// TIA Portal project "G INVERSION DE GIRO" (V11)

(* hardware
DEVICE "S7300/ET200 station_1"  SIMATIC 300-Station
   slot 0: "Perfil soporte_0"  Rail  6ES7 390-1***0-0AA0
   slot 2: "PLC_1"  CPU 313C-2 DP  6ES7 313-6CF03-0AB0  V2.6
      slot 0: "Interfaz MPI_1"  MPI
      slot 1: "Interfaz DP_1"  DP
      slot 2: "DI16/DO16_1"  DI16/DO16
      slot 4: "Contaje_1"  Counter
*)

// ===== PLC "PLC_1"  CPU 313C-2 DP =====

VAR_GLOBAL   // PLC tag table "Tabla de variables estándar"
   "Tag_1" AT %A0.0 : Bool;
   "Tag_2" AT %A0.1 : Bool;
   "Tag_3" AT %A0.2 : Bool;
   "Tag_4" AT %E0.0 : Bool;
   "Tag_5" AT %E0.1 : Bool;
   "Tag_6" AT %E0.2 : Bool;
   "Tag_7" AT %T0 : Timer;
   "Tag_8" AT %M0.0 : Bool;
END_VAR

DATA_BLOCK "INVERSION DE GIRO_DB"   // DB1
{ S7_Optimized_Access := 'FALSE' }
VERSION : 0.1
// stored: InstanceOfName INVERSION DE GIRO
"INVERSION DE GIRO"
BEGIN
   SWITCH[0] := 16#0;
   SW_SQTS[0] := 16#3;
   SW_SQTS[1] := 16#0;
   SW_SQTS[2] := 16#1;
   SW_SQTS[3] := 16#2;
   TVX[0] := 16#1;
   TTX[0] := 16#1;
   TSX[0] := 16#1;
   S00X[0] := 16#1;
   SOFFX[0] := 16#1;
   SONX[0] := 16#1;
   SAX[0] := 16#1;
   SERRX[0] := 16#1;
   SMX[0] := 16#1;
   S0X[0] := 16#1;
   S1X[0] := 16#1;
   SINI[0] := 16#2;
   SINI[1] := 16#1;
   LSTT[3] := 16#1;
   LSTT[4] := 16#1;
   ATAJ[1] := 16#1;
   ATAJ[2] := 16#2;
   ATAJ[3] := 16#3;
   ATAJ[4] := 16#4;
   ATAB[1] := 16#2;
   ATAB[2] := 16#1;
   ATAB[3] := 16#3;
   ATAB[4] := 16#4;
   PSTT[1] := 16#1;
   PSTT[2] := 16#1;
   PSTT[3] := 16#2;
   PSTT[4] := 16#3;
   NSTT[0] := 16#1;
   NSTT[1] := 16#2;
   NSTT[2] := 16#3;
   NSTT[3] := 16#1;
   NSTT[4] := 16#1;
   ASSJ[1] := 16#1;
   ASSJ[2] := 16#2;
   ASSJ[3] := 16#3;
   ASSB[1] := 16#1;
   ASSB[2] := 16#2;
   ASSB[3] := 16#3;
   PTTS[1] := 16#0;
   PTTS[2] := 16#1;
   PTTS[3] := 16#2;
   NTTS[1] := 16#1;
   NTTS[2] := 16#3;
   NTTS[3] := 16#4;
END_DATA_BLOCK

FUNCTION_BLOCK "INVERSION DE GIRO"   // FB1, GRAPH
{ S7_Optimized_Access := 'FALSE' }
VERSION : 0.1
   VAR_INPUT
      OFF_SQ : Bool := false;   // Desconectar cadena
      INIT_SQ : Bool := false;   // Poner cadena en estado inicial
      ACK_EF : Bool := false;   // Acusar todos los errores y fallos
      S_PREV : Bool := false;   // Mostrar la etapa anterior en el parámetro S_NO
      S_NEXT : Bool := false;   // Mostrar la etapa siguiente en el parámetro S_NO
      SW_AUTO : Bool := false;   // Modo automático
      SW_TAP : Bool := false;   // Semiautomático/continuar con transición
      SW_TOP : Bool := false;   // Semiautomático/transición ignorada
      SW_MAN : Bool := false;   // Modo manual
      S_SEL : Int := 0;   // Seleccionar la etapa que debe mostrarse en S_NO
      S_ON : Bool := false;   // Activar la etapa del parámetro S_NO
      S_OFF : Bool := false;   // Desactivar el incremento presente en el parámetro S_NO
      T_PUSH : Bool := false;   // Habilitar transición en modo semiautomático
      "MARCHA DERECHA" : Bool;
      "MARCHA IZQUIERDA" : Bool;
      PARO : Bool;
   END_VAR
   VAR_OUTPUT
      S_NO : Int := 0;   // Número de etapa
      S_MORE : Bool := false;   // Existen más etapas que pueden mostrarse en S_NO.
      S_ACTIVE : Bool := false;   // El incremento presente en el parámetro S_NO está activo
      ERR_FLT : Bool := false;   // Error de grupo interlock o supervisión
      AUTO_ON : Bool := false;   // Modo automático activado
      TAP_ON : Bool := false;   // Modo semiautomático/etapa con transición activada
      TOP_ON : Bool := false;   // Modo semiautomático/Ignorar transición activado
      MAN_ON : Bool := false;   // Modo manual activado
      "GIRO DERECHA" : Bool;
      "GIRO IZQUIERDA" : Bool;
   END_VAR
   VAR
      SWITCH : Array [0..0]of DWord;
      SW_SQTS : Array [0..3]of Byte;
      SW_ADDR : Word := 16#A;
      G7T_0 : GraphTransition;
      DERECHA : GraphTransition;
      IZQUIERDA : GraphTransition;
      "PARO D" : GraphTransition;
      "PARO I" : GraphTransition;
      G7S_0 : GraphStep;
      REPOSO : GraphStep;
      "M.D." : GraphStep;
      "M.I." : GraphStep;
      PRE_CRIT : Array [0..0]of DWord;
      POST_CRIT : Array [0..0]of DWord;
      TVX : Array [0..4]of Byte;
      TTX : Array [0..4]of Byte;
      TSX : Array [0..2]of Byte;
      S00X : Array [0..2]of Byte;
      SOFFX : Array [0..2]of Byte;
      SONX : Array [0..2]of Byte;
      SAX : Array [0..2]of Byte;
      SERRX : Array [0..4]of Byte;
      SMX : Array [0..4]of Byte;
      S0X : Array [0..4]of Byte;
      S1X : Array [0..4]of Byte;
      S_DISPLAY : Int;   // Indicación interna del parámetro de salida S_NO
      S_SEL_OLD : Int;   // Valor anterior en S_SEL
      S_DISPIDX : Byte;   // Índice de la etapa presente en S_NO
      T_DISPIDX : Byte;   // Índice de la transición presente en T_NO
      MOPEDGE : Struct
         AUTO : Bool := false;
         MAN : Bool := false;
         TAP : Bool := false;
         TOP : Bool := false;
         ACK_S : Bool := false;
         REG_S : Bool := false;
         T_PREV : Bool := false;
         T_NEXT : Bool := false;
         LOCK : Bool := false;
         SUP : Bool := false;
         ACKREQ : Bool := false;
         SSKIP : Bool := false;
         OFF : Bool := false;
         INIT : Bool := false;
         HALT : Bool := false;
         TMS_HALT : Bool := false;
         OPS_ZERO : Bool := false;
         SACT_DISP : Bool := false;
         SEF_DISP : Bool := false;
         SALL_DISP : Bool := false;
         S_PREV : Bool := false;
         S_NEXT : Bool := false;
         S_SELOK : Bool := false;
         S_ON : Bool := false;
         S_OFF : Bool := false;
         T_PUSH : Bool := false;
         REG : Bool := false;
         ACK : Bool := false;
         IL_PERM : Bool := false;
         T_PERM : Bool := false;
         ILP_MAN : Bool := false;
      END_STRUCT;
      MOP : Struct   // Modo de operación
         AUTO : Bool := true;   // Estado: modo automático
         MAN : Bool := false;   // Estado: modo manual
         TAP : Bool := false;   // Estado: semiautomático/continuar con transición
         TOP : Bool := false;   // Estado: semiautomático/transición ignorada
         ACK_S : Bool := false;   // Solicitud: acusar la etapa presente en el parámetro S_NO
         REG_S : Bool := false;   // Solicitud: registrar la etapa presente en el parámetro S_NO
         T_PREV : Bool := false;   // Solicitud: mostrar la transición anterior válida en el parámetro T_NO
         T_NEXT : Bool := false;   // Solicitud: mostrar la siguiente transición válida en el parámetro T_NO
         LOCK : Bool := true;   // Estado: ejecución de interlock activada
         SUP : Bool := true;   // Estado: ejecución de supervisión activada
         ACKREQ : Bool := true;   // Estado: acuse requerido
         SSKIP : Bool := false;   // Estado: "Saltar etapas" activado
         OFF : Bool := false;   // Solicitud: desactivar todas las etapas
         INIT : Bool := true;   // Solicitud: poner cadena en estado inicial
         HALT : Bool := false;   // Estado: la cadena no continúa
         TMS_HALT : Bool := false;   // Estado: todos los temporizadores internos detenidos
         OPS_ZERO : Bool := false;   // Estado: todos los operandos ejecutados con N, L, D puestos a 0
         SACT_DISP : Bool := true;   // Estado: mostrar sólo etapas activas
         SEF_DISP : Bool := false;   // Estado: mostrar sólo etapas erróneas y defectuosas
         SALL_DISP : Bool := false;   // Estado: mostrar todas las etapas
         S_PREV : Bool := false;   // Solicitud: mostrar la etapa anterior en el parámetro S_NO
         S_NEXT : Bool := false;   // Solicitud: Indicar etapa siguiente en el parámetro S_NO
         S_SELOK : Bool := false;   // Solicitud: mostrar en el parámetro S_NO el número de la etapa presente en el parámetro S_SEL
         S_ON : Bool := false;   // Solicitud: activar la etapa presente en el parámetro S_NO
         S_OFF : Bool := false;   // Solicitud: desactivar la etapa presente en el parámetro S_NO
         T_PUSH : Bool := false;   // Solicitud: habilitar transición
         REG : Bool := false;   // Solicitud: registrar todos los errores de interlock y supervisión
         ACK : Bool := false;   // Solicitud: acusar todos los errores de interlock y supervisión
         IL_PERM : Bool := false;   // Estado: ejecución permanente de todos los interlocks
         T_PERM : Bool := false;   // Estado: ejecución permanente de todas las transiciones
         ILP_MAN : Bool := false;   // Estado: ejecución permanente de todos los interlocks en modo manual
      END_STRUCT;
      TICKS : Struct   // Ciclos de tiempo
         DELTA : Time := T#0ms;   // Diferencia de tiempo entre dos ciclos
         OLD : Time := T#0ms;   // Estado de contador cíclico 10 ms en el último ciclo
         NEW : Time := T#0ms;   // Estado de contador cíclico 10 ms en este ciclo
      END_STRUCT;
      SQ_FLAGS : Struct   // Marcas de cadena
         ERR_FLT : Bool := false;   // Error de grupo interlock y supervisión
         ERROR : Bool := false;   // Error de grupo Interlock
         FAULT : Bool := false;   // Error de grupo Supervisión
         RT_FAIL : Bool := false;   // Error en tiempo de ejecución
         NO_SNO : Bool := false;   // No se ha encontrado el número de etapa solicitado
         NF_OFL : Bool := false;   // Desbordamiento: demasiadas solicitudes ON u OFF
         SA_OFL : Bool := false;   // Desbordamiento: demasiadas etapas activas
         TV_OFL : Bool := false;   // Desbordamiento: demasiadas transiciones válidas
         MSG_OFL : Bool := false;   // Desbordamiento: los recursos del sistema no son suficientes para ALARM_S
         NO_SWI : Bool := false;   // No conmutar en este ciclo
         CYC_OP : Bool := false;   // Ejecución cíclica de la cadena tras la inicialización
         AS_MSG : Bool := true;   // Avisos en tiempo de ejecución activados o desactivados por instrucción
         AS_SEND : Bool := false;   // Enviar avisos de WR_USMSG o sólo registrarlos en el búfer de diagnóstico
         SQ_BUSY : Bool := false;   // Marca de flanco interna para ejecución de proceso
         SA_BUSY : Bool := false;   // Marca de flanco interna para ejecución de proceso
         AS_SIG : Bool := false;   // Marca de flanco para avisos de Alarm_S y Alarm_SQ
      END_STRUCT;
      S_PTR : DWord := 16#320;
      S_PTR2 : DWord := 16#0;
      S_PTR3 : DWord := 16#8F0;
      S_PTR4 : DWord := 16#8C0;
      T_PTR : DWord := 16#890;
      C_AR2 : DWord := 16#0;
      M_FBDB : DWord := 16#10000;
      M_SNO : Word := 16#0;
      M_EVID : Word := 16#0;
      M_EVIL : C_Alarm_s;
      M_EVSV : C_Alarm_s;
      M_EV : DWord := 16#800;
      CRIT : Array [0..31]of Bool;
      S_START : Byte := 16#0;
      S_IDX : Byte := 16#0;
      S_INT : Int := 72;
      S_TMP : Byte := 16#0;
      T_START : Byte := 16#0;
      T_IDX : Byte := 16#0;
      T_TMP : Byte := 16#0;
      T_TMP2 : Byte := 16#00;
      TV_POT : Byte := 16#06;
      RETURN1 : Byte := 16#0;
      RETURN2 : Byte := 16#0;
      SINI : Array [0..2]of Byte;
      LSTT : Array [0..4]of Byte;
      ATAJ : Array [0..4]of Byte;
      ATAB : Array [0..4]of Byte;
      PSTT : Array [0..4]of Byte;
      NSTT : Array [0..4]of Byte;
      ASSJ : Array [0..3]of Byte;
      ASSB : Array [0..3]of Byte;
      PTTS : Array [0..3]of Byte;
      NTTS : Array [0..3]of Byte;
      PRE_CNT : Word := 16#1;
      POST_CNT : Word := 16#1;
      ADR_COND : Word := 16#0;
      MAX_TVAL : Byte := 16#3;
      MAX_SACT : Byte := 16#1;
      MAX_CRIT : Byte := 16#4;
      T_CNT : Byte := 16#4;
      SUP_CNT : Byte := 16#0;
      LOCK_CNT : Byte := 16#0;
      S_CNT : Byte := 16#3;
      SQ_CNT : Byte := 16#1;
      PRS_INPAR : DWord := 16#E000FEC8;
      PRS_OUTPAR : DWord := 16#E000800F;
      GC_FLAGS : Struct
         T_MACH : Byte := 16#EB;
         COND_ED : Byte := 16#E3;
         W_LEVEL : Byte := 16#D5;
         FB_IF : Byte := 16#FA;
         AS_MSG : Word := 16#202;
         SSB : Word := 16#108;
         DILG : Word := 16#1D6;
         ADDR_T0 : Word := 16#14;
         CRIT_AVAIL : Bool := false;
         SSKIP_AVAIL : Bool := true;
         SSKIP_ON : Bool := false;
         ACK_REQ : Bool := true;
         SYNC_AVAIL : Bool := true;
         ILP_MAN : Bool := false;
         SWM_LOCKED : Bool := false;
         SAVE_SW : Bool := true;
      END_STRUCT;
      G7_FBMARK : Byte := 16#3C;
      G7_RELEASE : Byte := 16#3C;
      G7_ID2 : Byte := 16#37;
      G7_ID1 : Byte := 16#47;
   END_VAR
   // SWITCH[0] := 16#0;
   // SW_SQTS[0] := 16#3;
   // SW_SQTS[1] := 16#0;
   // SW_SQTS[2] := 16#1;
   // SW_SQTS[3] := 16#2;
   // TVX[0] := 16#1;
   // TTX[0] := 16#1;
   // TSX[0] := 16#1;
   // S00X[0] := 16#1;
   // SOFFX[0] := 16#1;
   // SONX[0] := 16#1;
   // SAX[0] := 16#1;
   // SERRX[0] := 16#1;
   // SMX[0] := 16#1;
   // S0X[0] := 16#1;
   // S1X[0] := 16#1;
   // SINI[0] := 16#2;
   // SINI[1] := 16#1;
   // LSTT[3] := 16#1;
   // LSTT[4] := 16#1;
   // ATAJ[1] := 16#1;
   // ATAJ[2] := 16#2;
   // ATAJ[3] := 16#3;
   // ATAJ[4] := 16#4;
   // ATAB[1] := 16#2;
   // ATAB[2] := 16#1;
   // ATAB[3] := 16#3;
   // ATAB[4] := 16#4;
   // PSTT[1] := 16#1;
   // PSTT[2] := 16#1;
   // PSTT[3] := 16#2;
   // PSTT[4] := 16#3;
   // NSTT[0] := 16#1;
   // NSTT[1] := 16#2;
   // NSTT[2] := 16#3;
   // NSTT[3] := 16#1;
   // NSTT[4] := 16#1;
   // ASSJ[1] := 16#1;
   // ASSJ[2] := 16#2;
   // ASSJ[3] := 16#3;
   // ASSB[1] := 16#1;
   // ASSB[2] := 16#2;
   // ASSB[3] := 16#3;
   // PTTS[1] := 16#0;
   // PTTS[2] := 16#1;
   // PTTS[3] := 16#2;
   // NTTS[1] := 16#1;
   // NTTS[2] := 16#3;
   // NTTS[3] := 16#4;
BEGIN
END_FUNCTION_BLOCK

FUNCTION_BLOCK "ESTRELLA-TRIANGULO"   // FB2, GRAPH
{ S7_Optimized_Access := 'FALSE' }
VERSION : 0.1
   VAR_INPUT
      OFF_SQ : Bool := false;   // Desconectar cadena
      INIT_SQ : Bool := false;   // Poner cadena en estado inicial
      ACK_EF : Bool := false;   // Acusar todos los errores y fallos
      S_PREV : Bool := false;   // Mostrar la etapa anterior en el parámetro S_NO
      S_NEXT : Bool := false;   // Mostrar la etapa siguiente en el parámetro S_NO
      SW_AUTO : Bool := false;   // Modo automático
      SW_TAP : Bool := false;   // Semiautomático/continuar con transición
      SW_TOP : Bool := false;   // Semiautomático/transición ignorada
      SW_MAN : Bool := false;   // Modo manual
      S_SEL : Int := 0;   // Seleccionar la etapa que debe mostrarse en S_NO
      S_ON : Bool := false;   // Activar la etapa del parámetro S_NO
      S_OFF : Bool := false;   // Desactivar el incremento presente en el parámetro S_NO
      T_PUSH : Bool := false;   // Habilitar transición en modo semiautomático
      MARCHA : Bool;
      PARO : Bool;
   END_VAR
   VAR_OUTPUT
      S_NO : Int := 0;   // Número de etapa
      S_MORE : Bool := false;   // Existen más etapas que pueden mostrarse en S_NO.
      S_ACTIVE : Bool := false;   // El incremento presente en el parámetro S_NO está activo
      ERR_FLT : Bool := false;   // Error de grupo interlock o supervisión
      AUTO_ON : Bool := false;   // Modo automático activado
      TAP_ON : Bool := false;   // Modo semiautomático/etapa con transición activada
      TOP_ON : Bool := false;   // Modo semiautomático/Ignorar transición activado
      MAN_ON : Bool := false;   // Modo manual activado
      LINEA : Bool;
      ESTRELLA : Bool;
      TRIANGULO : Bool;
   END_VAR
   VAR
      S_DISPLAY : Int;   // Indicación interna del parámetro de salida S_NO
      S_SEL_OLD : Int;   // Valor anterior en S_SEL
      S_DISPIDX : Byte;   // Índice de la etapa presente en S_NO
      T_DISPIDX : Byte;   // Índice de la transición presente en T_NO
      MOP : Struct   // Modo de operación
         AUTO : Bool := true;   // Estado: modo automático
         MAN : Bool := false;   // Estado: modo manual
         TAP : Bool := false;   // Estado: semiautomático/continuar con transición
         TOP : Bool := false;   // Estado: semiautomático/transición ignorada
         ACK_S : Bool := false;   // Solicitud: acusar la etapa presente en el parámetro S_NO
         REG_S : Bool := false;   // Solicitud: registrar la etapa presente en el parámetro S_NO
         T_PREV : Bool := false;   // Solicitud: mostrar la transición anterior válida en el parámetro T_NO
         T_NEXT : Bool := false;   // Solicitud: mostrar la siguiente transición válida en el parámetro T_NO
         LOCK : Bool := true;   // Estado: ejecución de interlock activada
         SUP : Bool := true;   // Estado: ejecución de supervisión activada
         ACKREQ : Bool := true;   // Estado: acuse requerido
         SSKIP : Bool := false;   // Estado: "Saltar etapas" activado
         OFF : Bool := false;   // Solicitud: desactivar todas las etapas
         INIT : Bool := true;   // Solicitud: poner cadena en estado inicial
         HALT : Bool := false;   // Estado: la cadena no continúa
         TMS_HALT : Bool := false;   // Estado: todos los temporizadores internos detenidos
         OPS_ZERO : Bool := false;   // Estado: todos los operandos ejecutados con N, L, D puestos a 0
         SACT_DISP : Bool := true;   // Estado: mostrar sólo etapas activas
         SEF_DISP : Bool := false;   // Estado: mostrar sólo etapas erróneas y defectuosas
         SALL_DISP : Bool := false;   // Estado: mostrar todas las etapas
         S_PREV : Bool := false;   // Solicitud: mostrar la etapa anterior en el parámetro S_NO
         S_NEXT : Bool := false;   // Solicitud: Indicar etapa siguiente en el parámetro S_NO
         S_SELOK : Bool := false;   // Solicitud: mostrar en el parámetro S_NO el número de la etapa presente en el parámetro S_SEL
         S_ON : Bool := false;   // Solicitud: activar la etapa presente en el parámetro S_NO
         S_OFF : Bool := false;   // Solicitud: desactivar la etapa presente en el parámetro S_NO
         T_PUSH : Bool := false;   // Solicitud: habilitar transición
         REG : Bool := false;   // Solicitud: registrar todos los errores de interlock y supervisión
         ACK : Bool := false;   // Solicitud: acusar todos los errores de interlock y supervisión
         IL_PERM : Bool := false;   // Estado: ejecución permanente de todos los interlocks
         T_PERM : Bool := false;   // Estado: ejecución permanente de todas las transiciones
         ILP_MAN : Bool := false;   // Estado: ejecución permanente de todos los interlocks en modo manual
      END_STRUCT;
      TICKS : Struct   // Ciclos de tiempo
         DELTA : Time := T#0ms;   // Diferencia de tiempo entre dos ciclos
         OLD : Time := T#0ms;   // Estado de contador cíclico 10 ms en el último ciclo
         NEW : Time := T#0ms;   // Estado de contador cíclico 10 ms en este ciclo
      END_STRUCT;
      SQ_FLAGS : Struct   // Marcas de cadena
         ERR_FLT : Bool := false;   // Error de grupo interlock y supervisión
         ERROR : Bool := false;   // Error de grupo Interlock
         FAULT : Bool := false;   // Error de grupo Supervisión
         RT_FAIL : Bool := false;   // Error en tiempo de ejecución
         NO_SNO : Bool := false;   // No se ha encontrado el número de etapa solicitado
         NF_OFL : Bool := false;   // Desbordamiento: demasiadas solicitudes ON u OFF
         SA_OFL : Bool := false;   // Desbordamiento: demasiadas etapas activas
         TV_OFL : Bool := false;   // Desbordamiento: demasiadas transiciones válidas
         MSG_OFL : Bool := false;   // Desbordamiento: los recursos del sistema no son suficientes para ALARM_S
         NO_SWI : Bool := false;   // No conmutar en este ciclo
         CYC_OP : Bool := false;   // Ejecución cíclica de la cadena tras la inicialización
         AS_MSG : Bool := true;   // Avisos en tiempo de ejecución activados o desactivados por instrucción
         AS_SEND : Bool := false;   // Enviar avisos de WR_USMSG o sólo registrarlos en el búfer de diagnóstico
         SQ_BUSY : Bool := false;   // Marca de flanco interna para ejecución de proceso
         SA_BUSY : Bool := false;   // Marca de flanco interna para ejecución de proceso
         AS_SIG : Bool := false;   // Marca de flanco para avisos de Alarm_S y Alarm_SQ
      END_STRUCT;
      ARRANQUE : GraphTransition;
      REPOSO : GraphStep;
      "L-E." : GraphStep;
      TEMPORIZADO : GraphTransition;
   END_VAR
BEGIN
END_FUNCTION_BLOCK

ORGANIZATION_BLOCK "Main"   // OB1, LAD
TITLE = "Main Program Sweep (Cycle)"
{ S7_Optimized_Access := 'FALSE' }
VERSION : 0.1
   VAR_TEMP
      OB1_EV_CLASS : Byte;   // Bits 0-3 = 1 (Coming event), Bits 4-7 = 1 (Event class 1)
      OB1_SCAN_1 : Byte;   // 1 (Cold restart scan 1 of OB 1), 3 (Scan 2-n of OB 1)
      OB1_PRIORITY : Byte;   // Priority of OB Execution
      OB1_OB_NUMBR : Byte;   // 1 (Organization block 1, OB1)
      OB1_RESERVED_1 : Byte;   // Reserved for system
      OB1_RESERVED_2 : Byte;   // Reserved for system
      OB1_PREV_CYCLE : Int;   // Cycle time of previous OB1 scan (milliseconds)
      OB1_MIN_CYCLE : Int;   // Minimum cycle time of OB1 (milliseconds)
      OB1_MAX_CYCLE : Int;   // Maximum cycle time of OB1 (milliseconds)
      OB1_DATE_TIME : Date_And_Time;   // Date and time OB1 started
   END_VAR
BEGIN

REGION Network 1
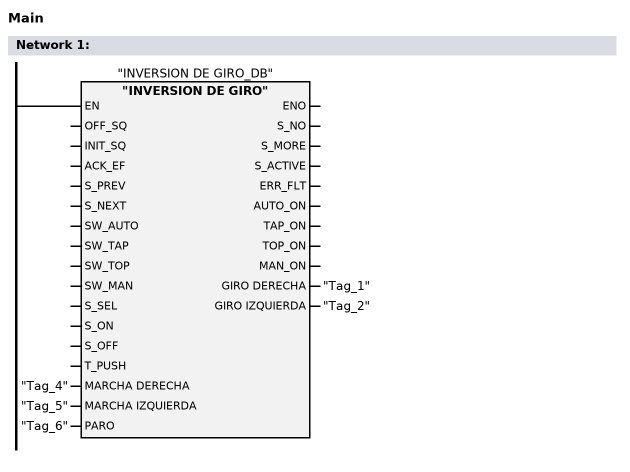
   RUNG wire#powerrail
      "INVERSION DE GIRO_DB"(OFF_SQ :=, INIT_SQ :=, ACK_EF :=, S_PREV :=, S_NEXT :=, SW_AUTO :=, SW_TAP :=, SW_TOP :=, SW_MAN :=, S_SEL :=, S_ON :=, S_OFF :=, T_PUSH :=, "MARCHA DERECHA" := "Tag_4", "MARCHA IZQUIERDA" := "Tag_5", PARO := "Tag_6", S_NO =>, S_MORE =>, S_ACTIVE =>, ERR_FLT =>, AUTO_ON =>, TAP_ON =>, TOP_ON =>, MAN_ON =>, "GIRO DERECHA" => "Tag_1", "GIRO IZQUIERDA" => "Tag_2")
   END_RUNG
   // the same network as SCL:
   "INVERSION DE GIRO_DB"("MARCHA DERECHA" := "Tag_4",   // "INVERSION DE GIRO"
                          "MARCHA IZQUIERDA" := "Tag_5",
                          PARO := "Tag_6",
                          "GIRO DERECHA" => "Tag_1",
                          "GIRO IZQUIERDA" => "Tag_2");
END_REGION
END_ORGANIZATION_BLOCK